(* IEC 61131-3 sources: eCockpitGit/test_project/src/%F%00 Library/%F%Common Functions/%F%String/%F%Normal/%F%Edit, 4 files *)

(* ---- %POU%FU_sDelete.st ---- *)
//This functions deletes a part of a string
// +-----------+----------+----------+-----------------------------------------------------------------------------------------------------------------------+
// |**Version**|**Author**| **Date** |**Changes**                                                                                                            |
// +-----------+----------+----------+-----------------------------------------------------------------------------------------------------------------------+
// | 1         | NSN      | 13-06-18 | Creation                                                                                                              |
// +-----------+----------+----------+-----------------------------------------------------------------------------------------------------------------------+
// | 1.1       | NSN      | 05-02-19 | Made dependant on big output version                                                                                  |
// +-----------+----------+----------+-----------------------------------------------------------------------------------------------------------------------+
FUNCTION FU_sDelete : STRING(255)
VAR_INPUT
	sStr		:STRING(255);		//Input String
	wLen		:WORD;				//Amount to delete
	wPos		:WORD;				//Position to delete from
END_VAR
(*%!%__DELIMITER__%!%*)
FU_sDeleteBIBO(sOut:= FU_sDelete,sStr:= sStr,wLen:= wLen,wPos:= wPos,wOutSize:= 255);

(* ---- %POU%FU_sDeleteRight.st ---- *)
//This functions deletes a part of a string values are counted from the right instead of the left
// +-----------+----------+----------+-----------------------------------------------------------------------------------------------------------------------+
// |**Version**|**Author**| **Date** |**Changes**                                                                                                            |
// +-----------+----------+----------+-----------------------------------------------------------------------------------------------------------------------+
// | 1         | NSN      | 22-02-19 | Creation                                                                                                              |
// +-----------+----------+----------+-----------------------------------------------------------------------------------------------------------------------+
FUNCTION FU_sDeleteRight : STRING(255)
VAR_INPUT
	sStr		:STRING(255);		//Input String
	wLen		:WORD;				//Amount to delete
	wPos		:WORD;				//Position to delete from
END_VAR
(*%!%__DELIMITER__%!%*)
FU_sDeleteRightBIBO(sOut:= FU_sDeleteRight, sStr:= sStr, wLen:= wLen,wPos:= wPos, wOutSize:= 255);

(* ---- %POU%FU_sMid.st ---- *)
//This functions extracts a part of a string
// +-----------+----------+----------+-----------------------------------------------------------------------------------------------------------------------+
// |**Version**|**Author**| **Date** |**Changes**                                                                                                            |
// +-----------+----------+----------+-----------------------------------------------------------------------------------------------------------------------+
// | 1         | NSN      | 13-06-18 | Creation                                                                                                              |
// +-----------+----------+----------+-----------------------------------------------------------------------------------------------------------------------+
// | 1.1       | NSN      | 05-02-19 | Made dependant on big output version                                                                                  |
// +-----------+----------+----------+-----------------------------------------------------------------------------------------------------------------------+
FUNCTION FU_sMid : STRING(255)
VAR_INPUT
	sStr		:STRING(255);		//Input String
	wLen		:WORD;				//Amount to copy
	wPos		:WORD;				//Position to copy from
END_VAR
(*%!%__DELIMITER__%!%*)
FU_sMidBIBO(sOut:= FU_sMid,sStr:= sStr,wLen:= wLen,wPos:= wPos,wOutSize:= 255);

(* ---- %POU%FU_sMidRight.st ---- *)
//This functions extracts a part of a string, values are counted from the right instead of the left
// +-----------+----------+----------+-----------------------------------------------------------------------------------------------------------------------+
// |**Version**|**Author**| **Date** |**Changes**                                                                                                            |
// +-----------+----------+----------+-----------------------------------------------------------------------------------------------------------------------+
// | 1         | NSN      | 22-02-19 | Creation                                                                                                              |
// +-----------+----------+----------+-----------------------------------------------------------------------------------------------------------------------+
FUNCTION FU_sMidRight : STRING(255)
VAR_INPUT
	sStr		:STRING(255);		//Input String
	wLen		:WORD;				//Amount to copy
	wPos		:WORD;				//Position to copy from
END_VAR
(*%!%__DELIMITER__%!%*)
FU_sMidRightBIBO(sOut:= FU_sMidRight,sStr:= sStr,wLen:= wLen,wPos:= wPos,wOutSize:= 255);
